Universal Robots PolyScope program: movep_61.urp

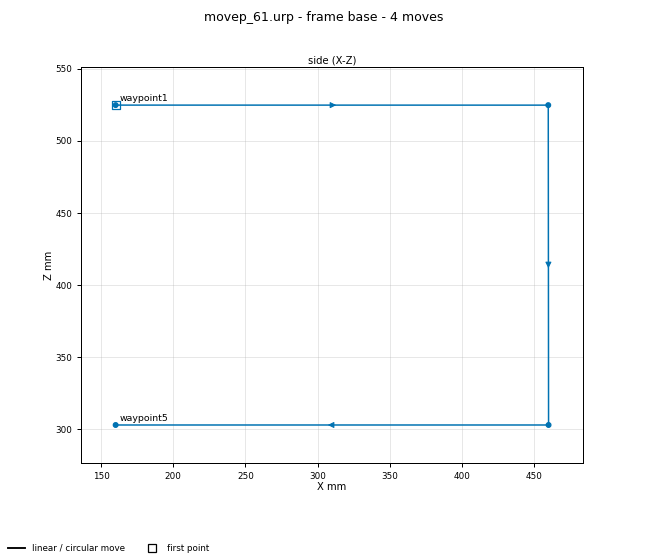
[picture p0: tool path of movep_61.urp in frame base, 4 of 4 moves have a stored position in this frame; points joined in program order, loops and branches not executed]
Program movep_61 (createdIn=3.2.19293 lastSavedIn=3.2.19293 directory=/programs installation=default robotSerialNumber=2015351391)
Calibrated DH parameters: a=[0.000352, -0.161198, -0.373486, 0.00005, 0.000049, 0]; d=[0.089268, 352.477598, -320.08558, -32.281492, 0.094939, 0.082518]; alpha=[1.570728, 0.001116, -0.003686, 1.571189, -1.570572, 0]; deltaTheta=[-0.000012, 1.181849, -1.491165, 0.309495, -0.000007, 0.000025]
Robot Program (runOnlyOnce=false motionType=MoveJ speed=1.047198 acceleration=1.396263 recalculateMotions=false)
  MoveP speed 250 mm/s, acceleration 1200 mm/s^2 (blendRadius=0.025 recalculateMotions=false) feature=Base
    Waypoint waypoint1: TCP in base x=160.014 y=198.812 z=524.837 mm, rx=-1.5849 ry=-0.1114 rz=-0.2807 rad; joints [73.38, -55.913, -125.557, 0.763, 100.407, -14.671] deg
    Waypoint waypoint3: TCP in base x=460.02 y=198.809 z=524.815 mm, rx=-1.5848 ry=-0.1115 rz=-0.2807 rad; joints [28.364, -98.879, -92.603, 10.03, 145.498, -15.62] deg
    Waypoint waypoint4: TCP in base x=460.231 y=198.899 z=303.004 mm, rx=-1.5851 ry=-0.1093 rz=-0.2825 rad; joints [28.343, -113.123, -110.59, 42.388, 145.472, -15.457] deg
    Waypoint waypoint5: TCP in base x=160.006 y=198.932 z=303.001 mm, rx=-1.5851 ry=-0.1094 rz=-0.2825 rad; joints [73.337, -75.201, -152.72, 47.232, 100.456, -14.549] deg
